gfCNCPoint5[29957] = {X 71.7013, Y 12.0458, Z -8.0000, A 0.000, B 0.000, C 0.000 }
gfCNCPoint5[29958] = {X 71.7021, Y 12.1868, Z -8.0000, A 0.000, B 0.000, C 0.000 }
gfCNCPoint5[29959] = {X 71.7016, Y 13.0911, Z -8.0000, A 0.000, B 0.000, C 0.000 }
gfCNCPoint5[29960] = {X 71.6387, Y 14.2141, Z -8.0000, A 0.000, B 0.000, C 0.000 }
gfCNCPoint5[29961] = {X 71.4717, Y 15.3264, Z -8.0000, A 0.000, B 0.000, C 0.000 }
gfCNCPoint5[29962] = {X 78.9573, Y 35.3501, Z -8.0000, A 0.000, B 0.000, C 0.000 }
gfCNCPoint5[29963] = {X 79.5722, Y 35.9628, Z -8.0000, A 0.000, B 0.000, C 0.000 }
gfCNCPoint5[29964] = {X 80.1416, Y 36.6180, Z -8.0000, A 0.000, B 0.000, C 0.000 }
gfCNCPoint5[29965] = {X 80.1416, Y 25.2445, Z -8.0000, A 0.000, B 0.000, C 0.000 }
gfCNCPoint5[29966] = {X 82.5416, Y 25.2445, Z -8.0000, A 0.000, B 0.000, C 0.000 }
gfCNCPoint5[29967] = {X 82.5417, Y 16.5233, Z -8.0000, A 0.000, B 0.000, C 0.000 }
gfCNCPoint5[29968] = {X 81.9009, Y 15.7818, Z -8.0000, A 0.000, B 0.000, C 0.000 }
gfCNCPoint5[29969] = {X 81.4212, Y 14.9271, Z -8.0000, A 0.000, B 0.000, C 0.000 }
gfCNCPoint5[29970] = {X 81.1220, Y 13.9938, Z -8.0000, A 0.000, B 0.000, C 0.000 }
gfCNCPoint5[29971] = {X 81.0153, Y 13.0196, Z -8.0000, A 0.000, B 0.000, C 0.000 }
gfCNCPoint5[29972] = {X 81.0151, Y 12.1868, Z -8.0000, A 0.000, B 0.000, C 0.000 }
gfCNCPoint5[29973] = {X 81.0160, Y 12.0923, Z -8.0000, A 0.000, B 0.000, C 0.000 }
gfCNCPoint5[29974] = {X 81.0187, Y 11.9978, Z -8.0000, A 0.000, B 0.000, C 0.000 }
gfCNCPoint5[29975] = {X 81.1325, Y 11.1229, Z -8.0000, A 0.000, B 0.000, C 0.000 }
gfCNCPoint5[29976] = {X 81.4019, Y 10.2827, Z -8.0000, A 0.000, B 0.000, C 0.000 }
gfCNCPoint5[29977] = {X 81.8181, Y 9.5048, Z -8.0000, A 0.000, B 0.000, C 0.000 }
gfCNCPoint5[29978] = {X 82.2192, Y 9.7686, Z -8.0000, A 0.000, B 0.000, C 0.000 }
gfCNCPoint5[29979] = {X 82.7660, Y 9.0935, Z -8.0000, A 0.000, B 0.000, C 0.000 }
gfCNCPoint5[29980] = {X 83.4348, Y 8.5389, Z -8.0000, A 0.000, B 0.000, C 0.000 }
gfCNCPoint5[29981] = {X 84.1996, Y 8.1266, Z -8.0000, A 0.000, B 0.000, C 0.000 }
gfCNCPoint5[29982] = {X 85.0305, Y 7.8726, Z -8.0000, A 0.000, B 0.000, C 0.000 }
gfCNCPoint5[29983] = {X 85.8951, Y 7.7868, Z -8.0000, A 0.000, B 0.000, C 0.000 }
gfCNCPoint5[29984] = {X 94.0497, Y 7.7868, Z -8.0000, A 0.000, B 0.000, C 0.000 }
gfCNCPoint5[29985] = {X 95.0288, Y 7.8971, Z -8.0000, A 0.000, B 0.000, C 0.000 }
gfCNCPoint5[29986] = {X 95.9588, Y 8.2226, Z -8.0000, A 0.000, B 0.000, C 0.000 }
gfCNCPoint5[29987] = {X 96.7930, Y 8.7468, Z -8.0000, A 0.000, B 0.000, C 0.000 }
gfCNCPoint5[29988] = {X 97.4897, Y 9.4435, Z -8.0000, A 0.000, B 0.000, C 0.000 }
gfCNCPoint5[29989] = {X 98.0139, Y 10.2777, Z -8.0000, A 0.000, B 0.000, C 0.000 }
gfCNCPoint5[29990] = {X 98.3394, Y 11.2077, Z -8.0000, A 0.000, B 0.000, C 0.000 }
gfCNCPoint5[29991] = {X 98.4497, Y 12.1868, Z -8.0000, A 0.000, B 0.000, C 0.000 }
gfCNCPoint5[29992] = {X 98.4494, Y 13.0233, Z -8.0000, A 0.000, B 0.000, C 0.000 }
gfCNCPoint5[29993] = {X 98.3725, Y 13.7986, Z -8.0000, A 0.000, B 0.000, C 0.000 }
gfCNCPoint5[29994] = {X 98.1599, Y 14.5482, Z -8.0000, A 0.000, B 0.000, C 0.000 }
gfCNCPoint5[29995] = {X 97.8185, Y 15.2486, Z -8.0000, A 0.000, B 0.000, C 0.000 }
gfCNCPoint5[29996] = {X 98.6471, Y 17.3116, Z -8.0000, A 0.000, B 0.000, C 0.000 }
gfCNCPoint5[29997] = {X 101.8766, Y 25.3093, Z -8.0000, A 0.000, B 0.000, C 0.000 }
gfCNCPoint5[29998] = {X 105.3627, Y 16.6199, Z -8.0000, A 0.000, B 0.000, C 0.000 }
gfCNCPoint5[29999] = {X 105.9232, Y 15.2215, Z -8.0000, A 0.000, B 0.000, C 0.000 }
gfCNCPoint5[30000] = {X 105.5852, Y 14.5144, Z -8.0000, A 0.000, B 0.000, C 0.000 }

ENDDAT
